// TIA Portal V16 export
// export: Created 2025-05-24T14:07:43.3676756Z, ExportSetting WithDefaults, DisplayName Totally Integrated Automation Portal, DisplayVersion V16, DisplayName TIA Portal Version Control Interface, DisplayVersion V16, DisplayName TIA Portal Openness, DisplayVersion V16, DisplayName STEP 7 Professional, DisplayVersion V16, DisplayName STEP 7 Safety, DisplayVersion V16, DisplayName WinCC Advanced, DisplayVersion V16
DATA_BLOCK "SwitchBlockAxisPosition_DB"   // DB39
VERSION : 0.1
// stored: AutoNumber true, InstanceOfName SwitchBlockAxisPosition, InstanceOfType FB
"SwitchBlockAxisPosition"
   // VAR_INPUT
   //    "Sensor Controlled" : Bool;
   //    Axis_Sensor_On_Position : Bool;
   //    Axis_Encoder_On_Position : Bool;
   // END_VAR
   // VAR_OUTPUT
   //    Axis_Measuring_Mode : Bool;
   // END_VAR
BEGIN
END_DATA_BLOCK
